// TIA Portal V19 export
DATA_BLOCK "PPrgArchive4"   // DB510
// stored: IsOnlyStoredInLoadMemory true, MemoryReserve 0, Namespace G
   VAR RETAIN
      PRG : Array[301..400] of "PPrg_Data";
   END_VAR
BEGIN
END_DATA_BLOCK
